(* PLC project , CODESYS GmbH CODESYS V3.5 *)

TYPE GoodType : int;
END_TYPE

TYPE GoodType : bool;
END_TYPE

PROGRAM Main

PROGRAM Main
END_PROGRAM
END_PROGRAM

FUNCTION_BLOCK Helper

FUNCTION_BLOCK Helper
END_FUNCTION_BLOCK
END_FUNCTION_BLOCK

PROGRAM LegacyDb

DATA_BLOCK LegacyDb
END_DATA_BLOCK
END_PROGRAM

CONFIGURATION Factory Config
  RESOURCE Line-1 ON PLC
  END_RESOURCE
END_CONFIGURATION
